// TIA Portal V17 export
// export: Created 2022-07-20T07:01:28.5313178Z, ExportSetting WithDefaults, DisplayName Totally Integrated Automation Portal, DisplayVersion V17, DisplayName TIA Portal Openness, DisplayVersion V17, DisplayName TIA Portal Version Control Interface, DisplayVersion V17, DisplayName SINAMICS Startdrive Advanced, DisplayVersion V17, DisplayName SINAMICS Startdrive G130, G150, S120, S150, SINAMICS MV, S210, DisplayVersion V17, DisplayName SINAMICS Startdrive G110M, G120, G120C, G120D, G120P, G115D, DisplayVersion V17, DisplayName STEP 7 Professional, DisplayVersion V17, DisplayName STEP 7 Safety, DisplayVersion V17, DisplayName WinCC Advanced, DisplayVersion V17
FUNCTION_BLOCK "FB10250_IfmAl2330"   // FB10250, LAD
{ S7_Optimized_Access := 'TRUE' }
VERSION : 0.1
// stored: AutoNumber false, IsIECCheckEnabled false, IsRetainMemResEnabled false, MemoryReserve 100, SetENOAutomatically false, UDAEnableTagReadback false
   VAR_INPUT
      PLC_In_Word_0 : Word;
      PLC_In_Word_2 : Word;
      PLC_In_Word_4 : Word;
      PLC_In_Word_6 : Word;
      "Active_X1.0_DO1" : Bool;
      "Active_X1.0_DO2" : Bool;
      "Active_X1.1_DO1" : Bool;
      "Active_X1.1_DO2" : Bool;
      "Active_X1.2_DO1" : Bool;
      "Active_X1.2_DO2" : Bool;
      "Active_X1.3_DO1" : Bool;
      "Active_X1.3_DO2" : Bool;
      "Active_X1.4_DO1" : Bool;
      "Active_X1.4_DO2" : Bool;
      "Active_X1.5_DO1" : Bool;
      "Active_X1.5_DO2" : Bool;
   END_VAR
   VAR_OUTPUT
      PLC_Out_Word_0 : Word;
      PLC_Out_Word_2 : Word;
      Id : UInt;
      DeviceStatus : UInt;
   END_VAR
   VAR
      DeviceStatusTemp : Byte;
   END_VAR
BEGIN

REGION Network 1 (SCL): Inputs Management
   //PLC In Word 0 Management

   //PLC In Word 2 Management

   //PLC In Word 4 Management

   //PLC In Word 6 Management
END_REGION

REGION Network 2 (SCL): Outputs Management
   //PLC Out Word 0 Management
   #PLC_Out_Word_0.%X0 := #"Active_X1.1_DO1";
   #PLC_Out_Word_0.%X1 := #"Active_X1.3_DO1";
   #PLC_Out_Word_0.%X2 := #"Active_X1.5_DO1";
   //#PLC_Out_Word_0.%X3 :=
   //#PLC_Out_Word_0.%X4 :=
   //#PLC_Out_Word_0.%X5 :=
   //#PLC_Out_Word_0.%X6 :=
   //#PLC_Out_Word_0.%X7 := 
   #PLC_Out_Word_0.%X8 := #"Active_X1.0_DO1";
   #PLC_Out_Word_0.%X9 := #"Active_X1.2_DO1";
   #PLC_Out_Word_0.%X10 := #"Active_X1.4_DO1";
   //#PLC_Out_Word_0.%X11 :=
   //#PLC_Out_Word_0.%X12 :=
   //#PLC_Out_Word_0.%X13 :=
   //#PLC_Out_Word_0.%X14 :=
   //#PLC_Out_Word_0.%X15 :=

   //PLC Out Word 2 Management
   #PLC_Out_Word_2.%X0 := #"Active_X1.1_DO2";
   #PLC_Out_Word_2.%X1 := #"Active_X1.3_DO2";
   #PLC_Out_Word_2.%X2 := #"Active_X1.5_DO2";
   //#PLC_Out_Word_2.%X3 :=
   //#PLC_Out_Word_2.%X4 :=
   //#PLC_Out_Word_2.%X5 :=
   //#PLC_Out_Word_2.%X6 :=
   //#PLC_Out_Word_2.%X7 :=
   #PLC_Out_Word_2.%X8 := #"Active_X1.0_DO2";
   #PLC_Out_Word_2.%X9 := #"Active_X1.2_DO2";
   #PLC_Out_Word_2.%X10 := #"Active_X1.4_DO2";
   //#PLC_Out_Word_2.%X11 :=
   //#PLC_Out_Word_2.%X12 :=
   //#PLC_Out_Word_2.%X13 :=
   //#PLC_Out_Word_2.%X14 :=
   //#PLC_Out_Word_2.%X15 :=
END_REGION
END_FUNCTION_BLOCK
